TYPE ST_AxisPersistent_back :
STRUCT

    iPositionAtShutdown : LREAL;
    bMovingAtShutdown   : BOOL;

END_STRUCT
END_TYPE

(* stored: Version 1.1.0.1, ProductVersion 3.1.4024.6
   DUT ST_AxisPersistent_back: Id {98d769cd-5416-4343-814a-f5a739d71156} *)
